PROGRAM Load_Mismatch_Not_Active
VAR
END_VAR

IF Stationary.LoadMismatchCheckTrigger.Q THEN
	
	//Told to pickup but have a load
	IF Otto.PickupLocation1 THEN

		IF Stationary.LoadPresent[2] AND Shuttle.GrabberLoaded[2] THEN 
		
			Stationary.LoadMismatchNotActive	:= TRUE;
		
		ELSE 
			
			Stationary.LoadMismatchNotActive	:= FALSE;
		
		END_IF
		
	ELSIF Otto.PickupLocation2 THEN  
	
		IF Stationary.LoadPresent[1] AND Shuttle.GrabberLoaded[1] THEN 
		
			Stationary.LoadMismatchNotActive	:= TRUE;
		
		ELSE 
			
			Stationary.LoadMismatchNotActive	:= FALSE;
		
		END_IF
		
	ELSIF Otto.DropoffLocation1 AND Stationary.LoadPresent[1] THEN 
		
		IF Stationary.LoadPresent[2] AND Shuttle.GrabberLoaded[2] THEN 
		
			Stationary.LoadMismatchNotActive	:= TRUE;
		
		ELSE 
			
			Stationary.LoadMismatchNotActive	:= FALSE;
		
		END_IF
		
	ELSIF Otto.DropoffLocation2 AND Stationary.LoadPresent[2] THEN  
	
		IF Stationary.LoadPresent[1] AND Shuttle.GrabberLoaded[1] THEN 
		
			Stationary.LoadMismatchNotActive	:= TRUE;
		
		ELSE 
			
			Stationary.LoadMismatchNotActive	:= FALSE;
		
		END_IF
		
	ELSE
		
		Stationary.LoadMismatchNotActive	:= FALSE;
		
	END_IF
	
END_IF

END_PROGRAM

(* stored: Version 1.1.0.1, ProductVersion 3.1.4024.9
   POU Load_Mismatch_Not_Active: Id {58cc65cb-53dc-4fc7-b598-e6175c22cc4e}, SpecialFunc None *)
